// TIA Portal V20 export
TYPE "LER_OEM_Data"
// stored: Access Published
   STRUCT
      FlexNet : "LER_FlexNet_Data";   // FlexNet
      PMC : "LER_PMC_Input_Data";   // PMC Data
   END_STRUCT;
END_TYPE
